// TIA Portal V20 export
TYPE "HMI_MonAn08"
   STRUCT
      PV_Hyst : Real := 1.0;   // PV - Alarm Hysteresis
      PV_Lim1 : Real;   // Limit 1
      PV_Lim2 : Real;   // Limit 2
      PV_Lim3 : Real;   // Limit 3
      PV_Lim4 : Real;   // Limit 4
      PV_Lim5 : Real;   // Limit 5
      PV_Lim6 : Real;   // Limit 6
      PV_Lim7 : Real;   // Limit 7
      PV_Lim8 : Real;   // Limit 8
      SmoothTi : Real;   // Smooth Time [s]
      SimPV : Real;   // Simulation Value
      RstOp : Bool;   // Reset Peak Values
      PV_OpScale : "ScaVal";   // PV - Bar Display Limits for OS
      PV_Unit : Int := 1001;   // Unit of PV
      DeadBand : Real;   // Dead band width
      TimeFactor : Int;   // Time Conversion Factor (0- Sec, 1- Min, 2- Hour)
      OnOp : Bool;   // 1=On Mode: On Mode by Operator
      OosOp : Bool;   // 1=Oos Mode: Oos Mode by Operator
      BypPVOp : Bool;   // 1 = Select bypass PV (via operator)
      RstBypOp : Bool;   // 1 = Reset bypass PV (via operator)
      PV_Out { ExternalWritable := 'False'} : Real;   // Process Value (Analog Output)
      PV_Out_ST { ExternalWritable := 'False'} : Byte := BYTE#16#80;   // PV_Out Signal Status
      PV_Grad { ExternalWritable := 'False'} : Real;   // PV - Gradient Value
      OS_PermOut { ExternalWritable := 'False'} : DWord := DWORD#16#FFFF_FFFF;   // Operator Permission: Output for OS
      OS1_PermOut { ExternalWritable := 'False'} : DWord := DWORD#16#FFFF_FFFF;   // Operator Permission: Output for OS
      OS_PermLog { ExternalWritable := 'False'} : DWord := DWORD#16#FFFF_FFFF;   // Operator Permission: Output for OS
      OS1_PermLog { ExternalWritable := 'False'} : DWord := DWORD#16#FFFF_FFFF;   // Operator Permission: Output for OS
      OpSt_Out { ExternalWritable := 'False'} : DWord;   // Enabled operator stations
      ST_Worst { ExternalWritable := 'False'} : Byte := 16#80;   // Worst Signal Status
      Status1 { ExternalWritable := 'False'} : DWord;   // Status1 Word
      Status2 { ExternalWritable := 'False'} : DWord;   // Status2 Word
      Status3 { ExternalWritable := 'False'} : DWord;   // Status3 Word
      Status4 { ExternalWritable := 'False'} : DWord;   // Status4 Word
      AlarmState { ExternalWritable := 'False'} : Word;   // Alarm Status for group display
   END_STRUCT;
END_TYPE
